{attribute 'strict'}
TYPE E_CognexCameraPutWatchStatus :
(
	WAITING_FOR_STATUS_CODE										:= 2,	
	THE_COMMAND_WAS_EXECUTED_SUCCESSFULLY						:= 1,
	UNRECOGNIZED_COMMAND 										:= 0,
	THE_INPUT_IS_INVALID_OR_HAS_EXCEEDED_15_BYTES_IN_LENGTH		:= -1,
	THE_COMMAND_COULD_NOT_BE_EXECUTED 							:= -2,
	USER_DOES_NOT_HAVE_FULL_ACCESS								:= -6
);
END_TYPE

(* stored: Version 1.1.0.1, ProductVersion 3.1.4024.12
   DUT E_CognexCameraPutWatchStatus: Id {197107f4-7afd-4a64-b3af-cc680245ede3} *)
